{library PUBLIC}
(* Station number type *)
TYPE StationType : INT(1..9);
END_TYPE

(* stored: Version 1.1.0.1, ProductVersion 3.1.4024.2
   EnumerationTextList StationType: Id {3e0b7e05-545d-4dc5-8d3e-569989a31c1d} *)
